FUNCTION_BLOCK AR2_TO_AR (* Composite FB for convert bidirectional AR2 to unidirectional AR *)
  (* Standard: 61499-2; Function: AR2_BIDIR forwards its incoming (EO1) side out as a plain unidirectional signal via AR_OUT. AR_IN publishes its value onto the outgoing (EI1) side of AR2_BIDIR.; Description: Copyright (c) 2026 HR Agrartechnik GmbH This program and the accompanying materials are made available under the terms of the Eclipse Public License 2.0 which is available at https://www.eclipse.org/legal/epl-2.0/ SPDX-License-Identifier: EPL-2.0 *)
  (* Version 1.0, 2026-08-31, Franz Höpfinger, HR Agrartechnik GmbH, Initial Version *)
  PACKAGE adapter::conversion::bidirectional;
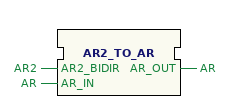
  SOCKETS
    AR2_BIDIR : adapter::types::bidirectional::AR2; (* Adapter Input: bidirectional tap, incoming side forwarded to AR_OUT, outgoing side driven by AR_IN *)
    AR_IN : adapter::types::unidirectional::AR; (* Adapter Input: unidirectional source *)
  END_SOCKETS
  PLUGS
    AR_OUT : adapter::types::unidirectional::AR; (* Adapter Output: mirrors AR2_BIDIR's incoming (indication) side *)
  END_PLUGS
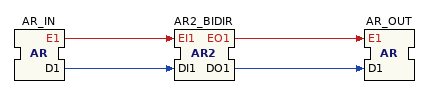
  EVENT_CONNECTIONS
    AR2_BIDIR.EO1 TO AR_OUT.E1;
    AR_IN.E1 TO AR2_BIDIR.EI1;
  END_CONNECTIONS
  DATA_CONNECTIONS
    AR2_BIDIR.DO1 TO AR_OUT.D1;
    AR_IN.D1 TO AR2_BIDIR.DI1;
  END_CONNECTIONS
END_FUNCTION_BLOCK
